Universal Robots PolyScope program: 31-pallet_working.urp

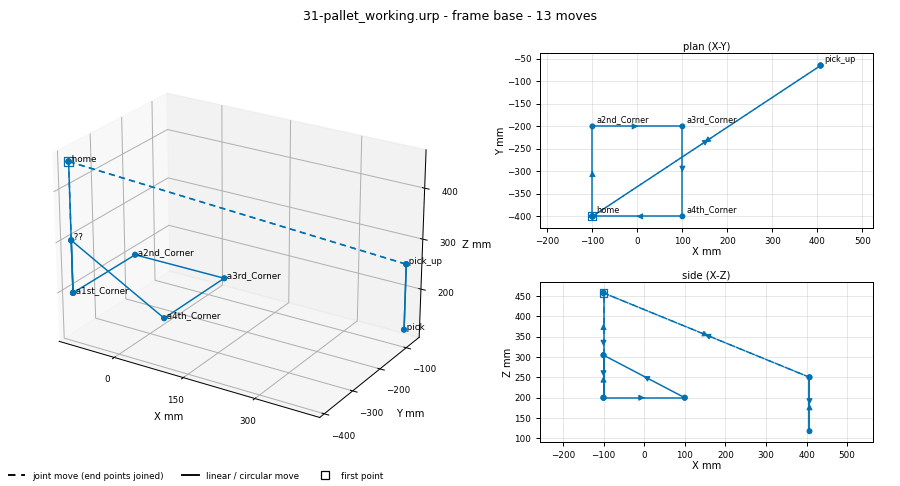
[picture p0: tool path of 31-pallet_working.urp in frame base, 13 of 13 moves have a stored position in this frame; points joined in program order, loops and branches not executed]
ProgramRoot directory=/home/ur/ursim-3.1/programs/basic training/31-pallet_working; kinematics=(a=[0, -0.425, -0.39225, 0, 0, 0], d=[0.08916, 0, 0, 0.10915, 0.09465, 0.0823], alpha=[1.5708, 0, 0, 1.5708, -1.5708, 0], deltaTheta=[0, 0, 0, 0, 0, 0], status=notInitialized); lastSavedInVersion=(project__name=Polyscope, major__version=3, minor__version=1, svn__revision=17195, build__date=Mar 11 2015, 13:02:28); name=31-pallet_working; programVersion=(project__name=Polyscope, major__version=3, minor__version=1, svn__revision=17195, build__date=Mar 11 2015, 13:02:28); robotEnvironmentFileName=default; serialNumberRobot=2014350001
  BeforeStart description=COMMAND_SEQUENCE_BEFORE_PROGRAM_START; name=BeforeStart
    Move cartesianAcceleration=1.2; cartesianSpeed=0.25; jointAcceleration=1.3962634015954636; jointSpeed=1.0471975511965976; sharedProcessMoveBlendRadius=0.025; motionType=JOINT_SPACE
      Waypoint blendRadius=0.05; cartesianAcceleration=1.2; cartesianSpeed=0.25; jointAcceleration=1.3962634015954636; jointSpeed=1.0471975511965976; nextMotionTime=2.0; stoppoint=true; useSharedBlendParameter=true; useSharedParameters=true; outputFlangePose=(pos=(x=-0.09999997057421518, y=-0.3999999686887875, z=0.4579999250079655), rot=(x=-0.0012210995541772555, y=3.116276478707302, z=0.03889232095780964)); position=TCP in base x=-100 y=-400 z=458 mm, rx=-0.0012 ry=3.1163 rz=0.0389 rad; joints [-88.988, -78.472, -96.118, -96.816, 91.461, 0.95] deg; positionType=FIXED_POSITION; waypointPoseInFeatureCoordinates=(pos=(x=-0.09999996879204003, y=-0.4000000219136234, z=0.4579998917979392), rot=(x=-0.001221102455289841, y=3.1162764786834214, z=0.03889232092108521)); name=home
    Assignment expr=5; operatorValueType=INTEGER; valueSource=EXPRESSION; variable=0
  MainProgram cartesianAcceleration=1.2; cartesianSpeed=0.25; jointAcceleration=1.3962634015954636; jointSpeed=1.0471975511965976; sharedProcessMoveBlendRadius=0.025; motionType=JOINT_SPACE
    Pallet patternSequenceNode=(MotionDefiningNode=(default=(cartesianAcceleration=1.2, cartesianSpeed=0.25, jointAcceleration=1.3962634015954636, jointSpeed=1.0471975511965976, recalculateMotions=false, sharedProcessMoveBlendRadius=0.025, motionType=CARTESIAN_SPACE)), AnchoredSequenceNode=(default=(name=托盘序列)))
      Pattern cartesianAcceleration=1.2; cartesianSpeed=0.25; jointAcceleration=1.3962634015954636; jointSpeed=1.0471975511965976; sharedProcessMoveBlendRadius=0.025; motionType=CARTESIAN_SPACE; dimensionality=4; firstAxisCount=6; secondAxisCount=4; thirdAxisCount=5; variable=0
        Waypoint blendRadius=0.05; cartesianAcceleration=1.2; cartesianSpeed=0.25; jointAcceleration=1.3962634015954636; jointSpeed=1.0471975511965976; nextMotionTime=2.0; stoppoint=true; useSharedBlendParameter=true; useSharedParameters=true; outputFlangePose=(pos=(x=-0.09999996906618717, y=-0.4000000540284308, z=0.19999996092213332), rot=(x=-0.0012210995541673518, y=3.116276478707373, z=0.03889232095778311)); position=TCP in base x=-100 y=-400 z=200 mm, rx=-0.0012 ry=3.1163 rz=0.0389 rad; joints [-88.988, -88.3, -127.491, -55.614, 91.461, 0.95] deg; positionType=FIXED_POSITION; waypointPoseInFeatureCoordinates=(pos=(x=-0.09999996819589951, y=-0.40000005265404437, z=0.1999999632555712), rot=(x=-0.001221102455286822, y=3.1162764786834214, z=0.03889232092108498)); name=a1st_Corner
        Waypoint blendRadius=0.05; cartesianAcceleration=1.2; cartesianSpeed=0.25; jointAcceleration=1.3962634015954636; jointSpeed=1.0471975511965976; nextMotionTime=2.0; stoppoint=true; useSharedBlendParameter=true; useSharedParameters=true; outputFlangePose=(pos=(x=-0.10000000337734316, y=-0.19999996438828968, z=0.19999998792032328), rot=(x=-0.001220853457287143, y=3.1162765026745656, z=0.038892110509023116)); position=TCP in base x=-100 y=-200 z=200 mm, rx=-0.0012 ry=3.1163 rz=0.0389 rad; joints [-87.972, -51.697, -148.925, -70.758, 91.486, 1.966] deg; positionType=FIXED_POSITION; waypointPoseInFeatureCoordinates=(pos=(x=-0.1000000033773473, y=-0.1999999639802142, z=0.1999999879203018), rot=(x=-0.0012208534573265933, y=3.1162765026745864, z=0.03889211050910507)); name=a2nd_Corner
        Waypoint blendRadius=0.05; cartesianAcceleration=1.2; cartesianSpeed=0.25; jointAcceleration=1.3962634015954636; jointSpeed=1.0471975511965976; nextMotionTime=2.0; stoppoint=true; useSharedBlendParameter=true; useSharedParameters=true; outputFlangePose=(pos=(x=0.10000003065018509, y=-0.19999997679949647, z=0.20000002024918062), rot=(x=-0.001220905866788091, y=3.116276536036987, z=0.03889203442944378)); position=TCP in base x=100 y=-200 z=200 mm, rx=-0.0012 ry=3.1163 rz=0.0389 rad; joints [-35.055, -51.443, -149.443, -68.76, 91.996, 54.906] deg; positionType=FIXED_POSITION; waypointPoseInFeatureCoordinates=(pos=(x=0.10000003093004557, y=-0.19999997679952106, z=0.20000002024915683), rot=(x=-0.0012209058668588384, y=3.1162765360370175, z=0.03889203442947606)); name=a3rd_Corner
        Waypoint blendRadius=0.05; cartesianAcceleration=1.2; cartesianSpeed=0.25; jointAcceleration=1.3962634015954636; jointSpeed=1.0471975511965976; nextMotionTime=2.0; stoppoint=true; useSharedBlendParameter=true; useSharedParameters=true; outputFlangePose=(pos=(x=0.10000008984722379, y=-0.39999992968002923, z=0.19999983963650697), rot=(x=-0.0012212291744449332, y=3.1162768257264872, z=0.038892683103488764)); position=TCP in base x=100 y=-400 z=200 mm, rx=-0.0012 ry=3.1163 rz=0.0389 rad; joints [-61.016, -88.295, -127.75, -54.511, 91.949, 28.93] deg; positionType=FIXED_POSITION; waypointPoseInFeatureCoordinates=(pos=(x=0.10000008984723645, y=-0.39999992995872546, z=0.19999983963652107), rot=(x=-0.0012212291743970486, y=3.116276825726508, z=0.038892683103293996)); name=a4th_Corner
      AnchoredSequence cartesianAcceleration=1.2; cartesianSpeed=0.25; jointAcceleration=1.3962634015954636; jointSpeed=1.0471975511965976; sharedProcessMoveBlendRadius=0.025; motionType=CARTESIAN_SPACE; anchoredWaypointNode=(PositionNode=(default=(blendRadius=0.05, cartesianAcceleration=1.2, cartesianSpeed=0.25, jointAcceleration=1.3962634015954636, jointSpeed=1.0471975511965976, nextMotionTime=2.0, specifyNextMotionTime=false, stoppoint=true, useSharedBlendParameter=true, useSharedParameters=true, positionType=FIXED_POSITION)), WaypointNode=(default=(name=模式点_1, relativeFromJointPositionVector=(joint=[nan, nan, nan, nan, nan, nan], isUndefined=true), relativeFromToolAxisAngle=(x=0.0, y=0.0, z=0.0), relativeFromToolPosition=(x=0.0, y=0.0, z=0.0)))); name=托盘序列
        Waypoint blendRadius=0.05; cartesianAcceleration=1.2; cartesianSpeed=0.25; jointAcceleration=1.3962634015954636; jointSpeed=1.0471975511965976; nextMotionTime=2.0; stoppoint=true; useSharedBlendParameter=true; useSharedParameters=true; outputFlangePose=(pos=(x=-0.09999997010097, y=-0.3999999954693952, z=0.30481860909342756), rot=(x=-0.0012210995542033655, y=3.1162764787073325, z=0.0388923209577967)); position=TCP in base x=-100 y=-400 z=304.819 mm, rx=-0.0012 ry=3.1163 rz=0.0389 rad; joints [-88.988, -80.778, -116.925, -73.702, 91.461, 0.95] deg; positionType=FIXED_POSITION; waypointPoseInFeatureCoordinates=(pos=(x=-0.09999996909892411, y=-0.40000000276892167, z=0.3048185500811591), rot=(x=-0.001221102455288116, y=3.1162764786834214, z=0.03889232092108509)); name=方式
        Waypoint blendRadius=0.05; cartesianAcceleration=1.2; cartesianSpeed=0.25; jointAcceleration=1.3962634015954636; jointSpeed=1.0471975511965976; nextMotionTime=2.0; stoppoint=true; useSharedBlendParameter=true; useSharedParameters=true; outputFlangePose=(pos=(x=-0.09999996906618717, y=-0.4000000540284308, z=0.19999996092213332), rot=(x=-0.001221099554167783, y=3.116276478707373, z=0.03889232095778312)); position=TCP in base x=-100 y=-400 z=200 mm, rx=-0.0012 ry=3.1163 rz=0.0389 rad; joints [-88.988, -88.3, -127.491, -55.614, 91.461, 0.95] deg; positionType=FIXED_POSITION; waypointPoseInFeatureCoordinates=(pos=(x=-0.09999996819589951, y=-0.40000005265404437, z=0.1999999632555712), rot=(x=-0.001221102455286822, y=3.1162764786834214, z=0.03889232092108498)); name=模式点_1
        Set 
        Wait 
        Waypoint blendRadius=0.05; cartesianAcceleration=1.2; cartesianSpeed=0.25; jointAcceleration=1.3962634015954636; jointSpeed=1.0471975511965976; nextMotionTime=2.0; stoppoint=true; useSharedBlendParameter=true; useSharedParameters=true; outputFlangePose=(pos=(x=-0.09999997010097, y=-0.3999999954693952, z=0.30481860909342756), rot=(x=-0.0012210995542033655, y=3.1162764787073325, z=0.0388923209577967)); position=TCP in base x=-100 y=-400 z=304.819 mm, rx=-0.0012 ry=3.1163 rz=0.0389 rad; joints [-88.988, -80.778, -116.925, -73.702, 91.461, 0.95] deg; positionType=FIXED_POSITION; waypointPoseInFeatureCoordinates=(pos=(x=-0.09999996909892411, y=-0.40000000276892167, z=0.3048185500811591), rot=(x=-0.001221102455288116, y=3.1162764786834214, z=0.03889232092108509)); name=退出
    Move cartesianAcceleration=1.2; cartesianSpeed=0.25; jointAcceleration=1.3962634015954636; jointSpeed=1.0471975511965976; sharedProcessMoveBlendRadius=0.025; motionType=JOINT_SPACE
      Waypoint blendRadius=0.05; cartesianAcceleration=1.2; cartesianSpeed=0.25; jointAcceleration=1.3962634015954636; jointSpeed=1.0471975511965976; nextMotionTime=2.0; stoppoint=true; useSharedBlendParameter=true; useSharedParameters=true; outputFlangePose=(pos=(x=-0.09999997057421518, y=-0.3999999686887875, z=0.4579999250079655), rot=(x=-0.0012210995541772555, y=3.116276478707302, z=0.03889232095780964)); position=TCP in base x=-100 y=-400 z=458 mm, rx=-0.0012 ry=3.1163 rz=0.0389 rad; joints [-88.988, -78.472, -96.118, -96.816, 91.461, 0.95] deg; positionType=FIXED_POSITION; waypointPoseInFeatureCoordinates=(pos=(x=-0.09999996879204003, y=-0.4000000219136234, z=0.4579998917979392), rot=(x=-0.001221102455289841, y=3.1162764786834214, z=0.03889232092108521)); name=home
      Waypoint blendRadius=0.05; cartesianAcceleration=1.2; cartesianSpeed=0.25; jointAcceleration=1.3962634015954636; jointSpeed=1.0471975511965976; nextMotionTime=2.0; stoppoint=true; useSharedBlendParameter=true; useSharedParameters=true; outputFlangePose=(pos=(x=0.40719162866152386, y=-0.06476752664969607, z=0.25038135230309055), rot=(x=2.315590396688657, y=-2.120233222113485, z=-0.05549569137880762)); position=TCP in base x=407.192 y=-64.768 z=250.381 mm, rx=2.3156 ry=-2.1202 rz=-0.0555 rad; joints [6.011, -83.984, -122.818, -64.604, 91.461, 0.95] deg; positionType=FIXED_POSITION; waypointPoseInFeatureCoordinates=(pos=(x=0.4071916281932563, y=-0.06476752666476945, z=0.25038140711775864), rot=(x=2.3155903964516824, y=-2.1202332224777143, z=-0.05549569138477739)); name=pick_up
    Move cartesianAcceleration=1.2; cartesianSpeed=0.25; jointAcceleration=1.3962634015954636; jointSpeed=1.0471975511965976; sharedProcessMoveBlendRadius=0.025; motionType=CARTESIAN_SPACE
      Waypoint blendRadius=0.05; cartesianAcceleration=1.2; cartesianSpeed=0.25; jointAcceleration=1.3962634015954636; jointSpeed=1.0471975511965976; nextMotionTime=2.0; stoppoint=true; useSharedBlendParameter=true; useSharedParameters=true; outputFlangePose=(pos=(x=0.4071914923292058, y=-0.06476754100508236, z=0.11756272126645136), rot=(x=2.3155903966880094, y=-2.120233222112948, z=-0.055495691379010295)); position=TCP in base x=407.191 y=-64.768 z=117.563 mm, rx=2.3156 ry=-2.1202 rz=-0.0555 rad; joints [6.011, -98.39, -133.227, -39.788, 91.461, 0.95] deg; positionType=FIXED_POSITION; waypointPoseInFeatureCoordinates=(pos=(x=0.4071914624463032, y=-0.06476754409000189, z=0.1175625989616466), rot=(x=2.3155902583603143, y=-2.1202331025077803, z=-0.05549593628812249)); name=pick
      Waypoint blendRadius=0.05; cartesianAcceleration=1.2; cartesianSpeed=0.25; jointAcceleration=1.3962634015954636; jointSpeed=1.0471975511965976; nextMotionTime=2.0; stoppoint=true; useSharedBlendParameter=true; useSharedParameters=true; outputFlangePose=(pos=(x=0.40719162866152386, y=-0.06476752664969607, z=0.25038135230309055), rot=(x=2.315590396688657, y=-2.120233222113485, z=-0.05549569137880762)); position=TCP in base x=407.192 y=-64.768 z=250.381 mm, rx=2.3156 ry=-2.1202 rz=-0.0555 rad; joints [6.011, -83.984, -122.818, -64.604, 91.461, 0.95] deg; positionType=FIXED_POSITION; waypointPoseInFeatureCoordinates=(pos=(x=0.4071916281932563, y=-0.06476752666476945, z=0.25038140711775864), rot=(x=2.3155903964516824, y=-2.1202332224777143, z=-0.05549569138477739)); name=pick_up
    Move cartesianAcceleration=1.2; cartesianSpeed=0.25; jointAcceleration=1.3962634015954636; jointSpeed=1.0471975511965976; sharedProcessMoveBlendRadius=0.025; motionType=JOINT_SPACE
      Waypoint blendRadius=0.05; cartesianAcceleration=1.2; cartesianSpeed=0.25; jointAcceleration=1.3962634015954636; jointSpeed=1.0471975511965976; nextMotionTime=2.0; stoppoint=true; useSharedBlendParameter=true; useSharedParameters=true; outputFlangePose=(pos=(x=-0.09999997057421518, y=-0.3999999686887875, z=0.4579999250079655), rot=(x=-0.0012210995541772555, y=3.116276478707302, z=0.03889232095780964)); position=TCP in base x=-100 y=-400 z=458 mm, rx=-0.0012 ry=3.1163 rz=0.0389 rad; joints [-88.988, -78.472, -96.118, -96.816, 91.461, 0.95] deg; positionType=FIXED_POSITION; waypointPoseInFeatureCoordinates=(pos=(x=-0.09999996879204003, y=-0.4000000219136234, z=0.4579998917979392), rot=(x=-0.001221102455289841, y=3.1162764786834214, z=0.03889232092108521)); name=home
